ABB RobotStudio station: WRITING_ARM.rspag

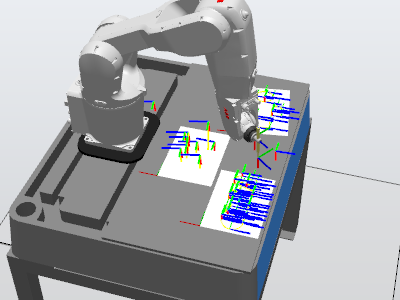
--- station ---
Station WRITING_ARM (saved by RobotStudio 25.2.11266.1)
Controller IRB1200_5_90, task T_ROB1: task frame (RAPID world) sits at (0, 233, 928) mm, rotated rx 0 ry 0 rz -90 deg in the station
Controller IRB1200_5_90
  mechanical unit ROB_1: IRB1200_5_90_STD_03, 6 joints, base frame (0, 0, 0) mm
Layout (positions relative to the parent item):
  - IRB1200_5_90_STD_03 [mechanism, from %ABB.RobotStudio.Models.IRB1200%\IRB1200_5_90_STD_03.rslib] at (0, 233, 928) mm, rotated rx 0 ry 0 rz -90 deg; joint values [0.0065, 1.0987, 0.3284, 0.6578, -1.4182, 0.0048] (rad or m)
  - Hardware [part], size 1120 x 955 x 931 mm
  - Pen for irb1200 [part] at (-45.84, -337.72, 1087.36) mm, rotated rx -157.43 ry 84.26 rz -14.37 deg, size 168 x 34 x 40 mm
Attachment: Pen for irb1200 is attached to IRB1200_5_90_STD_03 / Link6
Targets, tools, work objects and paths stored in the station and not in the controller backup, written as RAPID:
! task T_ROB1
MODULE Module1
  CONST robtarget LetterD40:=[[144,52,150],[0.0604561,0.734897,0.0624824,-0.672582],[-1,1,-1,1],[9E+09,9E+09,9E+09,9E+09,9E+09,9E+09]];
ENDMODULE


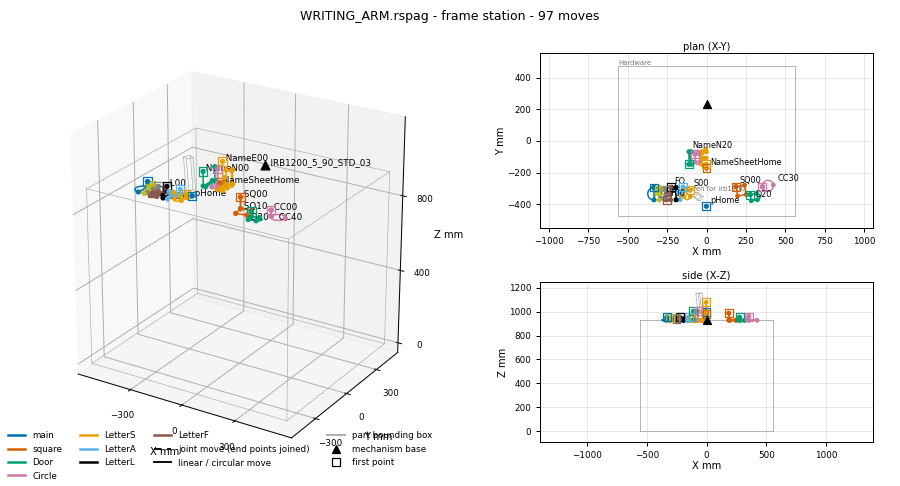
[picture p0: tool path of WRITING_ARM.rspag in frame station, 97 of 97 moves have a stored position in this frame; points joined in program order, loops and branches not executed]
--- Controller Data/IRB1200_5_90/RAPID/TASK1/PROGMOD/Module1.mod ---
MODULE Module1
	TASK PERS tooldata toolPen:=[TRUE,[[100,0,20],[1,0,0,0]],[0.1,[50,0,10],[1,0,0,0],0,0,0]];
	CONST robtarget pHome:=[[646.63,-1.2,67.59],[0.729459,0.00625806,0.683985,-0.00374601],[-1,0,0,1],[9E+09,9E+09,9E+09,9E+09,9E+09,9E+09]];
	TASK PERS wobjdata Shape_Sheet:=[FALSE,TRUE,"",[[455.474,135.551,0.105134],[0.000000814,0.0872218,-0.996189,0.000002429]],[[0,0,0],[1,0,0,0]]];
	LOCAL PERS robtarget SQ10:=[[-74.95,38.5,-0.01],[0.680832,0.0673549,-0.726353,0.0658941],[0,0,0,1],[9E+09,9E+09,9E+09,9E+09,9E+09,9E+09]];
	LOCAL PERS robtarget SQ20:=[[-74.95,93.41,-0.01],[0.680832,0.0673547,-0.726353,0.0658941],[0,0,-1,1],[9E+09,9E+09,9E+09,9E+09,9E+09,9E+09]];
	LOCAL PERS robtarget SQ30:=[[-134.85,93.45,-0.01],[0.680832,0.0673547,-0.726353,0.0658941],[0,0,-1,1],[9E+09,9E+09,9E+09,9E+09,9E+09,9E+09]];
	LOCAL PERS robtarget SQ40:=[[-134.85,38.56,-0.01],[0.680832,0.0673547,-0.726354,0.0658943],[0,0,-1,1],[9E+09,9E+09,9E+09,9E+09,9E+09,9E+09]];
	LOCAL PERS robtarget SQ00:=[[-74.95,38.5,-59.37],[0.680832,0.0673551,-0.726353,0.0658943],[0,0,-1,1],[9E+09,9E+09,9E+09,9E+09,9E+09,9E+09]];
	TASK PERS wobjdata Salford_Sheet:=[FALSE,TRUE,"",[[463.253,-387.169,0.139692],[0.0000021,0.0058094,-0.999983,0.000016811]],[[0,0,0],[1,0,0,0]]];
	LOCAL PERS robtarget SQ50:=[[-74.95,38.50,-0.01],[0.680832,0.0673549,-0.726353,0.0658941],[0,0,0,1],[9E+09,9E+09,9E+09,9E+09,9E+09,9E+09]];
	VAR robtarget D10:=[[-140.01,118.48,-0.01],[0.680832,0.067355,-0.726353,0.0658942],[0,0,-1,1],[9E+09,9E+09,9E+09,9E+09,9E+09,9E+09]];
	VAR robtarget D20:=[[-179.92,118.46,-0.01],[0.680832,0.067355,-0.726353,0.0658943],[0,0,-1,1],[9E+09,9E+09,9E+09,9E+09,9E+09,9E+09]];
	VAR robtarget D30:=[[-179.95,158,-0.01],[0.680831,0.0673549,-0.726354,0.0658945],[0,0,-1,1],[9E+09,9E+09,9E+09,9E+09,9E+09,9E+09]];
	VAR robtarget D50:=[[-140,158.49,-0.01],[0.680832,0.0673553,-0.726353,0.0658944],[0,0,-1,1],[9E+09,9E+09,9E+09,9E+09,9E+09,9E+09]];
	VAR robtarget D40:=[[-159.97,178.42,-0.01],[0.680832,0.067355,-0.726353,0.0658943],[0,0,-1,1],[9E+09,9E+09,9E+09,9E+09,9E+09,9E+09]];
	LOCAL PERS robtarget D00:=[[-140.01,118.48,-25],[0.680832,0.067355,-0.726353,0.0658943],[0,0,-1,1],[9E+09,9E+09,9E+09,9E+09,9E+09,9E+09]];
	VAR robtarget CC10:=[[-104.32,203.59,-0.01],[0.680833,0.0673548,-0.726353,0.065894],[0,0,-1,1],[9E+09,9E+09,9E+09,9E+09,9E+09,9E+09]];
	VAR robtarget CC30:=[[-104.98,273.41,-0.01],[0.680833,0.0673547,-0.726353,0.0658939],[0,0,-1,1],[9E+09,9E+09,9E+09,9E+09,9E+09,9E+09]];
	VAR robtarget CC20:=[[-70.08,238.52,-0.01],[0.680833,0.0673548,-0.726352,0.0658936],[0,0,-1,1],[9E+09,9E+09,9E+09,9E+09,9E+09,9E+09]];
	VAR robtarget CC40:=[[-139.68,238.64,-0.01],[0.680832,0.0673546,-0.726353,0.0658941],[0,0,-1,1],[9E+09,9E+09,9E+09,9E+09,9E+09,9E+09]];
	VAR robtarget CC00:=[[-105.24,203.48,-31.18],[0.680832,0.0673547,-0.726353,0.0658941],[0,0,-1,1],[9E+09,9E+09,9E+09,9E+09,9E+09,9E+09]];
	VAR robtarget S10:=[[-85.02,283.06,0.02],[0.683937,0.00797211,-0.729425,0.0102436],[-1,-1,-1,1],[9E+09,9E+09,9E+09,9E+09,9E+09,9E+09]];
	VAR robtarget S30:=[[-84.35,243.81,0.02],[0.683937,0.00797212,-0.729425,0.0102436],[-1,-1,-1,1],[9E+09,9E+09,9E+09,9E+09,9E+09,9E+09]];
	VAR robtarget S20:=[[-65.09,263.43,0.02],[0.683937,0.00797213,-0.729426,0.0102436],[-1,-1,-1,1],[9E+09,9E+09,9E+09,9E+09,9E+09,9E+09]];
	VAR robtarget S40:=[[-125.22,282.59,0.02],[0.683937,0.00797211,-0.729425,0.0102436],[-1,-1,0,1],[9E+09,9E+09,9E+09,9E+09,9E+09,9E+09]];
	VAR robtarget S60:=[[-124.94,243.82,0.02],[0.683936,0.0079722,-0.729426,0.0102435],[-1,-1,0,1],[9E+09,9E+09,9E+09,9E+09,9E+09,9E+09]];
	VAR robtarget S50:=[[-144.78,263.58,0.02],[0.683937,0.00797212,-0.729425,0.0102436],[-1,-1,0,1],[9E+09,9E+09,9E+09,9E+09,9E+09,9E+09]];
	VAR robtarget S70:=[[-113.17,232.46,-25.08],[0.683937,0.0079722,-0.729426,0.0102436],[-1,-1,0,1],[9E+09,9E+09,9E+09,9E+09,9E+09,9E+09]];
	VAR robtarget S00:=[[-85.02,283.06,-18.59],[0.683937,0.00797212,-0.729425,0.0102436],[-1,-1,-1,1],[9E+09,9E+09,9E+09,9E+09,9E+09,9E+09]];
	VAR robtarget S80:=[[-85.02,283.06,-18.59],[0.683937,0.00797212,-0.729425,0.0102436],[-1,-1,-1,1],[9E+09,9E+09,9E+09,9E+09,9E+09,9E+09]];
	VAR robtarget S90:=[[-124.94,243.82,-25.08],[0.683936,0.00797229,-0.729426,0.0102435],[-1,-1,0,1],[9E+09,9E+09,9E+09,9E+09,9E+09,9E+09]];
	VAR robtarget A10:=[[-64.96,238.12,0.02],[0.683936,0.00797236,-0.729426,0.0102434],[-1,-1,-1,1],[9E+09,9E+09,9E+09,9E+09,9E+09,9E+09]];
	VAR robtarget A20:=[[-144.8,218.39,0.02],[0.683936,0.00797249,-0.729427,0.0102434],[-1,-1,0,1],[9E+09,9E+09,9E+09,9E+09,9E+09,9E+09]];
	VAR robtarget A30:=[[-64.92,199.06,0.02],[0.683935,0.0079727,-0.729428,0.0102432],[-1,-1,-1,1],[9E+09,9E+09,9E+09,9E+09,9E+09,9E+09]];
	VAR robtarget A40:=[[-95.37,206.26,0.02],[0.683934,0.0079728,-0.729428,0.0102432],[-1,-1,0,1],[9E+09,9E+09,9E+09,9E+09,9E+09,9E+09]];
	VAR robtarget A50:=[[-95.58,230.38,0.02],[0.683934,0.00797279,-0.729429,0.0102431],[-1,-1,0,1],[9E+09,9E+09,9E+09,9E+09,9E+09,9E+09]];
	VAR robtarget A60:=[[-79.18,183.2,-6.83],[0.683934,0.00797275,-0.729429,0.0102431],[-1,-1,0,1],[9E+09,9E+09,9E+09,9E+09,9E+09,9E+09]];
	VAR robtarget A70:=[[-77.34,202.81,-6.83],[0.683934,0.00797262,-0.729428,0.0102432],[-1,-1,0,1],[9E+09,9E+09,9E+09,9E+09,9E+09,9E+09]];
	VAR robtarget A80:=[[-95.58,230.38,0.02],[0.683934,0.00797278,-0.729429,0.0102431],[-1,-1,0,1],[9E+09,9E+09,9E+09,9E+09,9E+09,9E+09]];
	VAR robtarget L10:=[[-65.25,163.53,0.02],[0.683937,0.0079723,-0.729425,0.0102434],[-1,-1,0,1],[9E+09,9E+09,9E+09,9E+09,9E+09,9E+09]];
	VAR robtarget L20:=[[-65.59,192.96,0.02],[0.683937,0.00797226,-0.729425,0.0102435],[-1,-1,-1,1],[9E+09,9E+09,9E+09,9E+09,9E+09,9E+09]];
	VAR robtarget L30:=[[-144.68,192.93,0.02],[0.683937,0.00797228,-0.729425,0.0102434],[-1,-1,0,1],[9E+09,9E+09,9E+09,9E+09,9E+09,9E+09]];
	VAR robtarget L40:=[[-144.68,192.93,-13.74],[0.683937,0.00797234,-0.729425,0.0102435],[-1,-1,0,1],[9E+09,9E+09,9E+09,9E+09,9E+09,9E+09]];
	VAR robtarget F00:=[[-144,134.28,-13.74],[0.683937,0.00797238,-0.729425,0.0102436],[-1,-1,0,1],[9E+09,9E+09,9E+09,9E+09,9E+09,9E+09]];
	VAR robtarget F10:=[[-144.44,128.46,0.02],[0.683937,0.00797217,-0.729426,0.0102435],[-1,-1,0,1],[9E+09,9E+09,9E+09,9E+09,9E+09,9E+09]];
	VAR robtarget F20:=[[-144.86,158.4,0.02],[0.683938,0.00797196,-0.729425,0.0102438],[-1,-1,0,1],[9E+09,9E+09,9E+09,9E+09,9E+09,9E+09]];
	VAR robtarget F30:=[[-105.12,157.38,0.02],[0.683937,0.00797213,-0.729425,0.0102436],[-1,-1,0,1],[9E+09,9E+09,9E+09,9E+09,9E+09,9E+09]];
	VAR robtarget F40:=[[-104.62,133.57,0.03],[0.683937,0.00797249,-0.729425,0.0102433],[-1,-1,0,1],[9E+09,9E+09,9E+09,9E+09,9E+09,9E+09]];
	VAR robtarget F50:=[[-65.25,158.06,0.02],[0.683936,0.00797224,-0.729426,0.0102433],[-1,-1,0,1],[9E+09,9E+09,9E+09,9E+09,9E+09,9E+09]];
	VAR robtarget F43:=[[-104.7,143.69,-3.18],[0.683936,0.00797229,-0.729426,0.0102432],[-1,-1,0,1],[9E+09,9E+09,9E+09,9E+09,9E+09,9E+09]];
	VAR robtarget FO:=[[-65.25,158.06,-18.82],[0.683936,0.00797239,-0.729427,0.0102432],[-1,-1,0,1],[9E+09,9E+09,9E+09,9E+09,9E+09,9E+09]];
	VAR robtarget O10:=[[-80.98,122.87,0.03],[0.683938,0.00797188,-0.729425,0.0102437],[-1,-1,0,1],[9E+09,9E+09,9E+09,9E+09,9E+09,9E+09]];
	VAR robtarget O30:=[[-80.64,93.67,0.03],[0.683937,0.00797195,-0.729425,0.0102435],[-1,-1,0,1],[9E+09,9E+09,9E+09,9E+09,9E+09,9E+09]];
	VAR robtarget O20:=[[-65.13,108.44,0.03],[0.683937,0.00797184,-0.729425,0.0102435],[-1,-1,0,1],[9E+09,9E+09,9E+09,9E+09,9E+09,9E+09]];
	VAR robtarget O40:=[[-129.81,94,0.03],[0.683937,0.00797184,-0.729426,0.0102434],[-1,-1,0,1],[9E+09,9E+09,9E+09,9E+09,9E+09,9E+09]];
	VAR robtarget O60:=[[-129.95,123.3,0.03],[0.683937,0.00797177,-0.729425,0.0102436],[-1,-1,0,1],[9E+09,9E+09,9E+09,9E+09,9E+09,9E+09]];
	VAR robtarget O50:=[[-144.6,108.44,0.03],[0.683937,0.00797195,-0.729426,0.0102434],[-1,-1,0,1],[9E+09,9E+09,9E+09,9E+09,9E+09,9E+09]];
	VAR robtarget O00:=[[-79.37,123.77,-19.95],[0.683937,0.00797199,-0.729426,0.0102436],[-1,-1,0,1],[9E+09,9E+09,9E+09,9E+09,9E+09,9E+09]];
	VAR robtarget R00:=[[-78.89,82.53,-19.95],[0.683937,0.00797213,-0.729426,0.0102436],[-1,-1,0,1],[9E+09,9E+09,9E+09,9E+09,9E+09,9E+09]];
	VAR robtarget R10:=[[-65.14,88.27,0.03],[0.683937,0.0079722,-0.729425,0.0102437],[-1,-1,0,1],[9E+09,9E+09,9E+09,9E+09,9E+09,9E+09]];
	VAR robtarget R20:=[[-144.6,87.35,0.03],[0.683937,0.0079722,-0.729425,0.0102437],[-1,-1,0,1],[9E+09,9E+09,9E+09,9E+09,9E+09,9E+09]];
	VAR robtarget R40:=[[-104.97,87.81,0.03],[0.683938,0.00797212,-0.729425,0.0102438],[-1,-1,0,1],[9E+09,9E+09,9E+09,9E+09,9E+09,9E+09]];
	VAR robtarget R30:=[[-124.94,58.84,0.03],[0.683937,0.00797226,-0.729425,0.0102436],[-1,-1,0,1],[9E+09,9E+09,9E+09,9E+09,9E+09,9E+09]];
	VAR robtarget R50:=[[-105.11,79.24,0.03],[0.683938,0.00797211,-0.729425,0.0102438],[-1,-1,0,1],[9E+09,9E+09,9E+09,9E+09,9E+09,9E+09]];
	VAR robtarget R60:=[[-64.79,59.06,0.03],[0.683937,0.00797208,-0.729425,0.0102438],[-1,-1,0,1],[9E+09,9E+09,9E+09,9E+09,9E+09,9E+09]];
	VAR robtarget RD:=[[-65.49,54.94,-11.67],[0.683937,0.00797238,-0.729426,0.0102441],[-1,-1,0,1],[9E+09,9E+09,9E+09,9E+09,9E+09,9E+09]];
	VAR robtarget LetterD10:=[[-64.88,53.48,0.03],[0.683938,0.00797241,-0.729425,0.0102433],[-1,-1,0,1],[9E+09,9E+09,9E+09,9E+09,9E+09,9E+09]];
	VAR robtarget LetterD30:=[[-144.58,52.63,0.03],[0.683938,0.00797247,-0.729425,0.0102433],[-1,-1,0,1],[9E+09,9E+09,9E+09,9E+09,9E+09,9E+09]];
	VAR robtarget LetterD20:=[[-105.13,14.04,0.03],[0.683937,0.00797255,-0.729425,0.0102431],[-1,-1,0,1],[9E+09,9E+09,9E+09,9E+09,9E+09,9E+09]];
	TASK PERS wobjdata Name_Sheet:=[FALSE,TRUE,"",[[237.648,-193.171,-0.010023],[2.42058E-05,-0.00550317,0.999985,-8.40246E-05]],[[0,0,0],[1,0,0,0]]];
	CONST robtarget calibrage2:=[[237.72,-193.17,-0.01],[0.0604561,0.734898,0.0624825,-0.672582],[-1,1,0,1],[9E+09,9E+09,9E+09,9E+09,9E+09,9E+09]];
	CONST robtarget calibrage12:=[[234.47,103.82,0.01],[0.114089,0.697844,-0.11409,-0.69784],[0,2,0,1],[9E+09,9E+09,9E+09,9E+09,9E+09,9E+09]];
	CONST robtarget calibrage22:=[[238.93,-193.43,0.01],[0.114089,0.697844,-0.11409,-0.697841],[-1,1,0,1],[9E+09,9E+09,9E+09,9E+09,9E+09,9E+09]];
	CONST robtarget calibrage1:=[[447.59,-190.86,0.00],[0.0604573,0.734898,0.0624844,-0.672582],[-1,1,-1,1],[9E+09,9E+09,9E+09,9E+09,9E+09,9E+09]];
	CONST robtarget calibrage3:=[[234.38,103.76,-0.06],[0.0604561,0.734897,0.0624824,-0.672582],[0,2,-1,1],[9E+09,9E+09,9E+09,9E+09,9E+09,9E+09]];
	CONST robtarget NameN10:=[[381,-112,0],[0.0604561,0.734897,0.0624824,-0.672582],[0,2,-1,1],[9E+09,9E+09,9E+09,9E+09,9E+09,9E+09]];
	CONST robtarget NameN20:=[[301,-112,0],[0.0604561,0.734897,0.0624824,-0.672582],[0,2,-1,1],[9E+09,9E+09,9E+09,9E+09,9E+09,9E+09]];
	CONST robtarget NameN30:=[[381,-97,0],[0.0604561,0.734897,0.0624824,-0.672582],[0,2,-1,1],[9E+09,9E+09,9E+09,9E+09,9E+09,9E+09]];
	CONST robtarget NameN40:=[[301,-97,0],[0.0604561,0.734897,0.0624824,-0.672582],[0,2,-1,1],[9E+09,9E+09,9E+09,9E+09,9E+09,9E+09]];
	CONST robtarget NameN50:=[[301,-97,75],[0.0604561,0.734897,0.0624824,-0.672582],[0,2,-1,1],[9E+09,9E+09,9E+09,9E+09,9E+09,9E+09]];
	CONST robtarget NameN00:=[[381,-112,75],[0.0604561,0.734897,0.0624824,-0.672582],[0,2,-1,1],[9E+09,9E+09,9E+09,9E+09,9E+09,9E+09]];
	CONST robtarget NameO10:=[[316,-72,0],[0.0604561,0.734897,0.0624824,-0.672582],[0,2,-1,1],[9E+09,9E+09,9E+09,9E+09,9E+09,9E+09]];
	CONST robtarget NameO20:=[[366,-72,0],[0.0604561,0.734897,0.0624824,-0.672582],[0,2,-1,1],[9E+09,9E+09,9E+09,9E+09,9E+09,9E+09]];
	CONST robtarget NameO30:=[[381,-57,0],[0.0604561,0.734897,0.0624824,-0.672582],[0,2,-1,1],[9E+09,9E+09,9E+09,9E+09,9E+09,9E+09]];
	CONST robtarget NameO40:=[[366,-42,0],[0.0604561,0.734897,0.0624824,-0.672582],[0,2,-1,1],[9E+09,9E+09,9E+09,9E+09,9E+09,9E+09]];
	CONST robtarget NameO50:=[[316,-42,0],[0.0604561,0.734897,0.0624824,-0.672582],[0,2,-1,1],[9E+09,9E+09,9E+09,9E+09,9E+09,9E+09]];
	CONST robtarget NameO60:=[[301,-57,0],[0.0604561,0.734897,0.0624824,-0.672582],[0,2,-1,1],[9E+09,9E+09,9E+09,9E+09,9E+09,9E+09]];
	CONST robtarget NameO00:=[[316,-72,75],[0.0604561,0.734897,0.0624824,-0.672582],[0,2,-1,1],[9E+09,9E+09,9E+09,9E+09,9E+09,9E+09]];
	CONST robtarget NameE10:=[[381,-2,0],[0.0604561,0.734897,0.0624824,-0.672582],[0,2,-1,1],[9E+09,9E+09,9E+09,9E+09,9E+09,9E+09]];
	CONST robtarget NameE20:=[[381,-32,0],[0.0604561,0.734897,0.0624824,-0.672582],[0,2,-1,1],[9E+09,9E+09,9E+09,9E+09,9E+09,9E+09]];
	CONST robtarget NameE30:=[[341,-32,0],[0.0604561,0.734897,0.0624824,-0.672582],[0,2,-1,1],[9E+09,9E+09,9E+09,9E+09,9E+09,9E+09]];
	CONST robtarget NameE40:=[[341,-2,0],[0.0604561,0.734897,0.0624824,-0.672582],[0,2,-1,1],[9E+09,9E+09,9E+09,9E+09,9E+09,9E+09]];
	CONST robtarget NameE50:=[[301,-32,0],[0.0604561,0.734897,0.0624824,-0.672582],[0,2,-1,1],[9E+09,9E+09,9E+09,9E+09,9E+09,9E+09]];
	CONST robtarget NameE60:=[[301,-2,0],[0.0604561,0.734897,0.0624824,-0.672582],[0,2,-1,1],[9E+09,9E+09,9E+09,9E+09,9E+09,9E+09]];
	CONST robtarget NameE00:=[[381,-2,150],[0.0604561,0.734897,0.0624824,-0.672582],[0,2,-1,1],[9E+09,9E+09,9E+09,9E+09,9E+09,9E+09]];
	CONST robtarget NameE21:=[[301,-82,50],[0.0604561,0.734897,0.0624824,-0.672582],[0,2,-1,1],[9E+09,9E+09,9E+09,9E+09,9E+09,9E+09]];
	CONST robtarget NameE41:=[[341,-17,50],[0.0604561,0.734897,0.0624824,-0.672582],[0,2,-1,1],[9E+09,9E+09,9E+09,9E+09,9E+09,9E+09]];
	CONST robtarget NameE70:=[[301,-2,75],[0.0604561,0.734897,0.0624824,-0.672582],[0,2,-1,1],[9E+09,9E+09,9E+09,9E+09,9E+09,9E+09]];
	CONST robtarget NameSheetHome:=[[406.67,-0.02,50.50],[2.8433E-05,0.707107,-2.84904E-05,-0.707107],[-1,1,0,1],[9E+09,9E+09,9E+09,9E+09,9E+09,9E+09]];
	CONST robtarget NameE80:=[[308,-29,75],[0.0604561,0.734897,0.0624824,-0.672582],[0,1,-1,1],[9E+09,9E+09,9E+09,9E+09,9E+09,9E+09]];
	CONST robtarget NameE90:=[[308,-29,0],[0.0604561,0.734897,0.0624824,-0.672582],[0,1,-1,1],[9E+09,9E+09,9E+09,9E+09,9E+09,9E+09]];
	CONST robtarget NameE100:=[[288,-5,0],[0.0604561,0.734897,0.0624824,-0.672582],[0,1,-1,1],[9E+09,9E+09,9E+09,9E+09,9E+09,9E+09]];
	CONST robtarget NameE110:=[[288,-5,75],[0.0604561,0.734897,0.0624824,-0.672582],[0,1,-1,1],[9E+09,9E+09,9E+09,9E+09,9E+09,9E+09]];
	VAR num Choose:=0;
	CONST string SalfordSheet:="";
	CONST string NameSheet:="";
	CONST string ShapeSheet:="";
	VAR num My_choice:=0;
	CONST string Which_sheet_do_you_want:="";
	VAR num MyChoice:=0;
	CONST robtarget A00:=[[-64.96,238.12,-25],[0.683937,0.00797242,-0.729426,0.0102433],[-1,-1,-1,1],[9E+09,9E+09,9E+09,9E+09,9E+09,9E+09]];
	CONST robtarget L00:=[[-65.25,163.53,-25],[0.683937,0.00797234,-0.729425,0.0102434],[-1,-1,0,1],[9E+09,9E+09,9E+09,9E+09,9E+09,9E+09]];
	CONST robtarget LetterD00:=[[-64.88,53.48,-25],[0.683938,0.00797259,-0.729425,0.0102434],[-1,-1,0,1],[9E+09,9E+09,9E+09,9E+09,9E+09,9E+09]];
    !***********************************************************
    !
    ! Module:  Module1
    !
    ! Description:
    !   <Insert description here>
    !
    ! Author: SUP926
    !
    ! Version: 1.0
    !
    !***********************************************************


    !***********************************************************
    !
    ! Procedure main
    !
    !   This is the entry point of your program
    !
    !***********************************************************
    PROC main()
        !Add your code here
        MoveJ pHome, v1000, z200, toolPen;
        TPErase;
        TPWrite "writing terminal";
        TPReadFK MyChoice, "which sheet", "Shape", "Salford", "Name", stEmpty, stEmpty;
        TEST MyChoice
        CASE 1:
        	Shape;
        CASE 2:
        	Salford;
        CASE 3:
        	Name;
        ENDTEST
        MoveJ pHome, v2500, z200, toolPen;
    ENDPROC
	PROC square()
		MoveJ SQ00, v1000, fine, toolPen\WObj:=Shape_Sheet;
		MoveL SQ10, v1000, fine, toolPen\WObj:=Shape_Sheet;
		MoveL SQ20, v1000, fine, toolPen\WObj:=Shape_Sheet;
		MoveL SQ30, v1000, fine, toolPen\WObj:=Shape_Sheet;
		MoveL SQ40, v1000, fine, toolPen\WObj:=Shape_Sheet;
		MoveL SQ10, v1000, fine, toolPen\WObj:=Shape_Sheet;
		MoveL SQ00, v1000, fine, toolPen\WObj:=Shape_Sheet;
	ENDPROC
	PROC Door()
		MoveJ D00, v500, z10, toolPen\WObj:=Shape_Sheet;
		MoveL D10, v1000, fine, toolPen\WObj:=Shape_Sheet;
		MoveL D20, v1000, fine, toolPen\WObj:=Shape_Sheet;
		MoveL D30, v1000, fine, toolPen\WObj:=Shape_Sheet;
		MoveC D40, D50, v1000, z1, toolPen\WObj:=Shape_Sheet;
		MoveL D10, v1000, fine, toolPen\WObj:=Shape_Sheet;
		MoveL D00, v1000, fine, toolPen\WObj:=Shape_Sheet;
	ENDPROC
	PROC Circle()
		MoveJ CC00, v500, z10, toolPen\WObj:=Shape_Sheet;
		MoveL CC10, v1000, fine, toolPen\WObj:=Shape_Sheet;
		MoveC CC20, CC30, v1000, fine, toolPen\WObj:=Shape_Sheet;
		MoveC CC40, CC10, v1000, fine, toolPen\WObj:=Shape_Sheet;
		MoveL CC00, v1000, z10, toolPen\WObj:=Shape_Sheet;
	ENDPROC
	PROC Shape()
		square;
		WaitTime 2;
		Door;
		WaitTime 2;
		Circle;
		WaitTime 2;
	ENDPROC
	PROC LetterS()
		MoveJ S00, v500, z10, toolPen\WObj:=Salford_Sheet;
		MoveL S10, v1000, fine, toolPen\WObj:=Salford_Sheet;
		MoveC S20, S30, v1000, z1, toolPen\WObj:=Salford_Sheet;
		MoveL S40, v1000, fine, toolPen\WObj:=Salford_Sheet;
		MoveC S50, S60, v1000, z1, toolPen\WObj:=Salford_Sheet;
		MoveL S70, v1000, z10, toolPen\WObj:=Salford_Sheet;
	ENDPROC
	PROC LetterA()
		MoveJ A00, v500, fine, toolPen\WObj:=Salford_Sheet;
		MoveL A10, v1000, fine, toolPen\WObj:=Salford_Sheet;
		MoveL A20, v1000, fine, toolPen\WObj:=Salford_Sheet;
		MoveL A30, v1000, fine, toolPen\WObj:=Salford_Sheet;
		MoveJ A70, v1000, z10, toolPen\WObj:=Salford_Sheet;
		MoveL A40, v1000, fine, toolPen\WObj:=Salford_Sheet;
		MoveL A50, v1000, fine, toolPen\WObj:=Salford_Sheet;
		MoveL A80, v1000, fine, toolPen\WObj:=Salford_Sheet;
		MoveJ A60, v1000, z10, toolPen\WObj:=Salford_Sheet;
	ENDPROC
	PROC LetterL()
		MoveJ L00, v500, z10, toolPen\WObj:=Salford_Sheet;
		MoveL L10, v1000, fine, toolPen\WObj:=Salford_Sheet;
		MoveL L20, v1000, fine, toolPen\WObj:=Salford_Sheet;
		MoveL L30, v1000, fine, toolPen\WObj:=Salford_Sheet;
		MoveJ L40, v1000, z10, toolPen\WObj:=Salford_Sheet;
	ENDPROC
	PROC LetterF()
		MoveJ F00, v500, z10, toolPen\WObj:=Salford_Sheet;
		MoveL F10, v1000, fine, toolPen\WObj:=Salford_Sheet;
		MoveL F20, v1000, fine, toolPen\WObj:=Salford_Sheet;
		MoveL F30, v1000, fine, toolPen\WObj:=Salford_Sheet;
		MoveL F40, v1000, fine, toolPen\WObj:=Salford_Sheet;
		MoveJ F43, v1000, z10, toolPen\WObj:=Salford_Sheet;
		MoveJ F30, v1000, fine, toolPen\WObj:=Salford_Sheet;
		MoveL F50, v1000, fine, toolPen\WObj:=Salford_Sheet;
		MoveL FO, v1000, z10, toolPen\WObj:=Salford_Sheet;
	ENDPROC
	PROC LetterO()
		MoveJ O00, v1000, z10, toolPen\WObj:=Salford_Sheet;
		MoveL O10, v1000, fine, toolPen\WObj:=Salford_Sheet;
		MoveC O20, O30, v1000, fine, toolPen\WObj:=Salford_Sheet;
		MoveL O40, v1000, z1, toolPen\WObj:=Salford_Sheet;
		MoveC O50, O60, v1000, fine, toolPen\WObj:=Salford_Sheet;
		MoveL O10, v1000, fine, toolPen\WObj:=Salford_Sheet;
		MoveJ O00, v1000, z10, toolPen\WObj:=Salford_Sheet;
	ENDPROC
	PROC LetterR()
		MoveJ R00, v1000, z10, toolPen\WObj:=Salford_Sheet;
		MoveL R10, v1000, fine, toolPen\WObj:=Salford_Sheet;
		MoveL R20, v1000, fine, toolPen\WObj:=Salford_Sheet;
		MoveC R30, R40, v1000, z1, toolPen\WObj:=Salford_Sheet;
		MoveJ R50, v1000, fine, toolPen\WObj:=Salford_Sheet;
		MoveL R60, v1000, fine, toolPen\WObj:=Salford_Sheet;
		MoveJ RD, v1000, z10, toolPen\WObj:=Salford_Sheet;
	ENDPROC
	PROC LetterD()
		MoveJ LetterD00, v500, fine, toolPen\WObj:=Salford_Sheet;
		MoveL LetterD10, v1000, fine, toolPen\WObj:=Salford_Sheet;
		MoveC LetterD20, LetterD30, v1000, fine, toolPen\WObj:=Salford_Sheet;
		MoveL LetterD10, v1000, fine, toolPen\WObj:=Salford_Sheet;
		MoveL LetterD00, v1000, z10, toolPen\WObj:=Salford_Sheet;
	ENDPROC
	PROC Salford()
		LetterS;
		LetterA;
		LetterL;
		LetterF;
		LetterO;
		LetterR;
		LetterD;
	ENDPROC
	PROC Name()
		MoveJ NameSheetHome, v1000, z60, toolPen;
		NameN;
		NameO;
		NameE;
	ENDPROC
	PROC NameN()
		MoveJ NameN00, v1000, z50, toolPen;
		MoveL NameN10, v1000, fine, toolPen;
		MoveL NameN20, v1000, fine, toolPen;
		MoveL NameN30, v1000, fine, toolPen;
		MoveL NameN40, v1000, fine, toolPen;
		MoveL NameN50, v1000, z50, toolPen;
	ENDPROC
	PROC NameO()
		MoveJ NameO00, v1000, z50, toolPen;
		MoveL NameO10, v1000, fine, toolPen;
		MoveL NameO20, v1000, fine, toolPen;
		MoveC NameO30, NameO40, v1000, fine, toolPen;
		MoveL NameO50, v1000, fine, toolPen;
		MoveC NameO60, NameO10, v1000, fine, toolPen;
		MoveL NameO00, v1000, fine, toolPen;
	ENDPROC
	PROC NameE()
		MoveJ NameE00, v1000, z20, toolPen;
		MoveL NameE10, v1000, fine, toolPen;
		MoveL NameE20, v1000, fine, toolPen;
		MoveL NameE30, v1000, fine, toolPen;
		MoveL NameE40, v1000, fine, toolPen;
		MoveL NameE41, v1000, z20, toolPen;
		MoveL NameE30, v1000, fine, toolPen;
		MoveL NameE50, v1000, fine, toolPen;
		MoveL NameE60, v1000, fine, toolPen;
		MoveL NameE70, v1000, z20, toolPen;
		MoveJ NameE80, v1000, z20, toolPen;
		MoveL NameE90, v1000, fine, toolPen;
		MoveL NameE100, v1000, fine, toolPen;
		MoveL NameE110, v1000, z50, toolPen;
	ENDPROC
ENDMODULE

--- Controller Data/IRB1200_5_90/RAPID/TASK1/SYSMOD/LINKEDM.sys ---
%%%
  VERSION:1
  LANGUAGE:ENGLISH
%%%

MODULE LINKEDM (SYSMODULE)

! FOLLOWER
!     Name of electronically linked follower axis used by operator at teach pendent.
      PERS string l_f_axis_name{5}       :=  ["",  "", "", "", ""];

!     Name of the mechanical unit for follower axis.
      PERS string l_f_mecunt_n{5}  :=  ["", "", "", "", ""];

!     Linked follower axis number in the mechanical unit (first axis in mech. unit is number 1).
      PERS num l_f_axis_no{5}      :=  [0,          0,   0,  0,  0];

! MASTER
!     Name of the mechanical unit for linked master axis.
      PERS string l_m_mecunt_n{5} :=  ["", "", "", "", ""];

!     Linked master axis number in the mechanical unit (first axis in mech. unit is number 1).
!     See axis number table in documentation for different master mechanical units.
      PERS num l_m_axis_no{5}     :=  [0,  0,  0,  0,  0];

! POSITION OFFSET
!     The increase of the allowed offset position between the master and follower
!     positions, used when starting AUTO mode. As soon as the offset is decreased
!     the old configurated parameter is used.
!     Example: 3 => the configurated value of allowed offset is increased 3 times.
      PERS num offset_ratio{5}       :=  [10,  10,   10,  10,  10];

! SPEED RATIO
!     Speed_ratio used in AUTO and JOG modes [ very_slow   slow    normal    fast]
!     Value 1 = max allowed manual speed.
      CONST num speed_ratio {20}      := [0.01, 0.01, 0.01, 0.01, 0.01,
                                          0.05, 0.05, 0.05, 0.05, 0.05,
                                          0.20, 0.20, 0.20, 0.20, 0.20,
                                          1.00, 1.00, 1.00, 1.00, 1.00];

! STEP SIZE
!     Displacement position used in JOG mode for each activation of positive or
!     negative movement.                  [very_short    short   normal   long]
!     Unit degees or meter.
      CONST num displacement {20}     := [0.001, 0.001, 0.001, 0.001, 0.001,
                                          0.005, 0.005, 0.005, 0.005, 0.005,
                                          0.020, 0.020, 0.020, 0.020, 0.020,
                                          0.100, 0.100, 0.100, 0.100, 0.100];


!-------------------------------------------------------------
 PROC Linked_m ()
      Linked_m_exe ;
 ENDPROC
ENDMODULE
